(* Logix 5000 project; controller SIMON Emulate 5570 rev 30.12; software revision 30.00 *)

TASK MainTask (periodic, rate 5000 ms, priority 1, watchdog 5000 ms) : MainProgram

MODULES
   Local : Emulate 5570 (ICP 2, rev 30.12)
       : vendor 1 type 0 code 15 (ICP 0, rev 1.1, Output RPI 50 ms)
END_MODULES

TYPE UDT_BA :
STRUCT
   AL : BOOL[128];
END_STRUCT
END_TYPE

PROGRAM MainProgram   (* main routine MainRoutine *)
VAR
   SCAN_CYCLE_TIME : DINT;
   Simon_Ciphertext : DINT[2,2];
   Simon_dec_i : DINT;
   Simon_dec_j : DINT;
   Simon_enc_i : DINT;
   Simon_enc_j : DINT;
   Simon_i : DINT;
   Simon_j : DINT;
   Simon_Plaintext : DINT[2,2];
   Simon_Rd_Max : DINT;
   Simon_Rotate_Result : DINT[2];
   Simon_Round_Keys : DINT[72,2];
   Simon_tmp1 : DINT[2];
   Simon_tmp2 : DINT[2];
   Simon_Ver : DINT;
   Simon_x : DINT[2];
   Simon_y : DINT[2];
END_VAR

ROUTINE MainRoutine   (* ladder *)
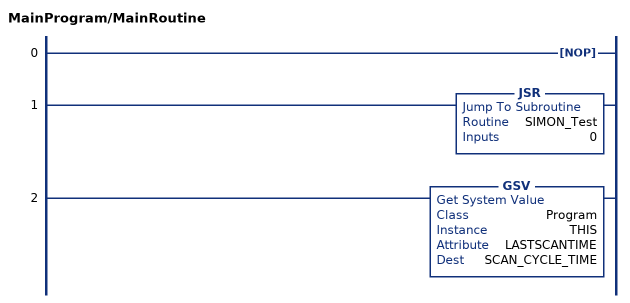
   0: NOP();
   1: JSR(SIMON_Test,0);
   2: GSV(Program,THIS,LASTSCANTIME,SCAN_CYCLE_TIME);
END_ROUTINE

ROUTINE SIMON_ClearKey   (* structured text *)
   Case Simon_Ver Of
   
   0,1,2:
   	For Simon_i:=0 to Simon_Rd_Max by 1 do
   		Simon_Round_Keys[Simon_i,0]:=0;
   	End_For;
   	Simon_tmp1[0]:=0;
   	Simon_tmp2[0]:=0;
   	Simon_Rotate_Result[0]:=0;
   3,4,5:
   	For Simon_i:=0 to Simon_Rd_Max by 1 do
   		Simon_Round_Keys[Simon_i,0]:=0;
   		Simon_Round_Keys[Simon_i,1]:=0;
   	End_For;
   	Simon_tmp1[0]:=0;
   	Simon_tmp1[1]:=0;
   	Simon_tmp2[0]:=0;
   	Simon_tmp2[1]:=0;
   	Simon_Rotate_Result[0]:=0;
   	Simon_Rotate_Result[1]:=0;
   End_Case;
   
   
END_ROUTINE

ROUTINE SIMON_Dec   (* structured text *)
   
   JSR(SIMON_Init);
   
   
   
   
   Case Simon_Ver Of
   
   0,1,2:
   	Simon_Plaintext[1,0]:=Simon_Ciphertext[0,0];
   	Simon_Plaintext[0,0]:=Simon_Ciphertext[1,0];
   
   	For Simon_i:=Simon_Rd_Max to 0 by -1 do
   		Simon_tmp2[0]:=Simon_Plaintext[0,0];  //for rotate
   		JSR(SIMON_Rotate_Left1);	//rotate based on Simon_Ciphertext[0,0]
   		Simon_tmp1[0]:= Simon_Rotate_Result[0];
   		Simon_Rotate_Result[0]:=0;
   
   		Simon_tmp2[0]:=Simon_Plaintext[0,0];  //for rotate
   		JSR(SIMON_Rotate_Left8);
   		Simon_tmp2[0]:=Simon_Rotate_Result[0];
   		Simon_tmp1[0]:= Simon_tmp1[0] AND Simon_tmp2[0];
   		Simon_Rotate_Result[0]:=0;
   
   		Simon_tmp2[0]:=Simon_Plaintext[0,0];  //for rotate
   		JSR(SIMON_Rotate_Left2);
   		Simon_tmp1[0]:= Simon_tmp1[0] XOR Simon_Rotate_Result[0];
   
   		Simon_tmp1[0]:= Simon_tmp1[0] XOR Simon_Round_Keys[Simon_i,0];
   
   		Simon_Plaintext[0,0]:= Simon_Plaintext[1,0] XOR Simon_tmp1[0];
   		Simon_Plaintext[1,0]:= Simon_tmp2[0];
   
   		Simon_Rotate_Result[0]:=0;
   
   	End_for;
   
   3,4,5:
   	Simon_Plaintext[1,0]:=Simon_Ciphertext[0,0];
   	Simon_Plaintext[1,1]:=Simon_Ciphertext[0,1];
   	Simon_Plaintext[0,0]:=Simon_Ciphertext[1,0];
   	Simon_Plaintext[0,1]:=Simon_Ciphertext[1,1];
   
   	For Simon_i:=Simon_Rd_Max to 0 by -1 do
   
   		Simon_tmp2[0]:=Simon_Plaintext[0,0];  //for rotate
   		Simon_tmp2[1]:=Simon_Plaintext[0,1];
   
   		JSR(SIMON_Rotate_Left1);	//rotate based on Simon_Ciphertext[0,0] and [0,1]
   		Simon_tmp1[0]:= Simon_Rotate_Result[0];
   		Simon_tmp1[1]:= Simon_Rotate_Result[1];
   
   		Simon_Rotate_Result[0]:=0;
   		Simon_Rotate_Result[1]:=0;
   
   		Simon_tmp2[0]:=Simon_Plaintext[0,0];
   		Simon_tmp2[1]:=Simon_Plaintext[0,1];
   		JSR(SIMON_Rotate_Left8);
   		Simon_tmp2[0]:=Simon_Rotate_Result[0];
   		Simon_tmp2[1]:=Simon_Rotate_Result[1];
   		Simon_tmp1[0]:= Simon_tmp1[0] AND Simon_tmp2[0];
   		Simon_tmp1[1]:= Simon_tmp1[1] AND Simon_tmp2[1];
   
   		Simon_tmp2[0]:=Simon_Plaintext[0,0];
   		Simon_tmp2[1]:=Simon_Plaintext[0,1];
   
   		Simon_Rotate_Result[0]:=0;
   		Simon_Rotate_Result[1]:=0;
   
   		JSR(SIMON_Rotate_Left2);
   		Simon_tmp1[0]:= Simon_tmp1[0] XOR Simon_Rotate_Result[0];
   		Simon_tmp1[1]:= Simon_tmp1[1] XOR Simon_Rotate_Result[1];
   
   		Simon_tmp1[0]:= Simon_tmp1[0] XOR Simon_Round_Keys[Simon_i,0];
   		Simon_tmp1[1]:= Simon_tmp1[1] XOR Simon_Round_Keys[Simon_i,1];
   
   
   		Simon_Plaintext[0,0]:= Simon_Plaintext[1,0] XOR Simon_tmp1[0];
   		Simon_Plaintext[0,1]:= Simon_Plaintext[1,1] XOR Simon_tmp1[1];
   
   		Simon_Plaintext[1,0]:= Simon_tmp2[0];
   		Simon_Plaintext[1,1]:= Simon_tmp2[1];
   
   		Simon_Rotate_Result[0]:=0;
   		Simon_Rotate_Result[1]:=0;
   
   	End_for;
   
   End_Case;
   
   
   
   
   
   
   JSR(SIMON_ClearKey);
   
   
   
   
   
   
   
   
END_ROUTINE

ROUTINE SIMON_Enc   (* structured text *)
   
   JSR(SIMON_Init);
   
   
   
   
   
   Case Simon_Ver Of
   
   0,1,2:
   	//Simon_Ciphertext[1,0]:=Simon_Plaintext[0,0];
   	//Simon_Ciphertext[0,0]:=Simon_Plaintext[1,0];
   
   	Simon_Ciphertext[0,0]:=Simon_Plaintext[1,0];
   	Simon_Ciphertext[1,0]:=Simon_Plaintext[0,0];
   
   	For Simon_i:=0 to Simon_Rd_Max by 1 do
   		Simon_tmp2[0]:=Simon_Ciphertext[0,0];  //for rotate
   		JSR(SIMON_Rotate_Left1);	//rotate based on Simon_Plaintext[0,0]
   		Simon_tmp1[0]:= Simon_Rotate_Result[0];
   		Simon_Rotate_Result[0]:=0;
   
   		Simon_tmp2[0]:=Simon_Ciphertext[0,0];  //for rotate
   		JSR(SIMON_Rotate_Left8);
   		Simon_tmp2[0]:=Simon_Rotate_Result[0];
   
   		Simon_tmp1[0]:= Simon_tmp1[0] AND Simon_tmp2[0];
   		Simon_Rotate_Result[0]:=0;
   
   		Simon_tmp2[0]:=Simon_Ciphertext[0,0];  //for rotate
   		JSR(SIMON_Rotate_Left2);
   		Simon_tmp1[0]:= Simon_tmp1[0] XOR Simon_Rotate_Result[0];
   
   		Simon_tmp1[0]:= Simon_tmp1[0] XOR Simon_Round_Keys[Simon_i,0];
   
   		Simon_Ciphertext[0,0]:= Simon_Ciphertext[1,0] XOR Simon_tmp1[0];
   		Simon_Ciphertext[1,0]:= Simon_tmp2[0];
   
   		Simon_Rotate_Result[0]:=0;
   
   	End_for;
   
   3,4,5:
   	Simon_Ciphertext[1,0]:=Simon_Plaintext[0,0];
   	Simon_Ciphertext[1,1]:=Simon_Plaintext[0,1];
   	Simon_Ciphertext[0,0]:=Simon_Plaintext[1,0];
   	Simon_Ciphertext[0,1]:=Simon_Plaintext[1,1];
   
   	For Simon_i:=0 to Simon_Rd_Max by 1 do
   
   		Simon_tmp2[0]:=Simon_Ciphertext[0,0];  //for rotate
   		Simon_tmp2[1]:=Simon_Ciphertext[0,1];
   
   		JSR(SIMON_Rotate_Left1);	//rotate based on Simon_Plaintext[0,0] and [0,1]
   		Simon_tmp1[0]:= Simon_Rotate_Result[0];
   		Simon_tmp1[1]:= Simon_Rotate_Result[1];
   
   		Simon_Rotate_Result[0]:=0;
   		Simon_Rotate_Result[1]:=0;
   
   		Simon_tmp2[0]:=Simon_Ciphertext[0,0];
   		Simon_tmp2[1]:=Simon_Ciphertext[0,1];
   		JSR(SIMON_Rotate_Left8);
   		Simon_tmp2[0]:=Simon_Rotate_Result[0];
   		Simon_tmp2[1]:=Simon_Rotate_Result[1];
   		Simon_tmp1[0]:= Simon_tmp1[0] AND Simon_tmp2[0];
   		Simon_tmp1[1]:= Simon_tmp1[1] AND Simon_tmp2[1];
   
   		Simon_Rotate_Result[0]:=0;
   		Simon_Rotate_Result[1]:=0;
   
   		Simon_tmp2[0]:=Simon_Ciphertext[0,0];
   		Simon_tmp2[1]:=Simon_Ciphertext[0,1];
   		JSR(SIMON_Rotate_Left2);
   		Simon_tmp1[0]:= Simon_tmp1[0] XOR Simon_Rotate_Result[0];
   		Simon_tmp1[1]:= Simon_tmp1[1] XOR Simon_Rotate_Result[1];
   
   		Simon_tmp1[0]:= Simon_tmp1[0] XOR Simon_Round_Keys[Simon_i,0];
   		Simon_tmp1[1]:= Simon_tmp1[1] XOR Simon_Round_Keys[Simon_i,1];
   
   
   		Simon_Ciphertext[0,0]:= Simon_Ciphertext[1,0] XOR Simon_tmp1[0];
   		Simon_Ciphertext[0,1]:= Simon_Ciphertext[1,1] XOR Simon_tmp1[1];
   
   		Simon_Ciphertext[1,0]:= Simon_tmp2[0];
   		Simon_Ciphertext[1,1]:= Simon_tmp2[1];
   
   		Simon_Rotate_Result[0]:=0;
   		Simon_Rotate_Result[1]:=0;
   
   	End_for;
   
   End_Case;
   
   
   
   
   
   JSR(SIMON_ClearKey);
   
   
   
   
   
   
END_ROUTINE

ROUTINE SIMON_Init   (* structured text *)
   CASE Simon_Ver Of
   	0:
   		Simon_Rd_Max:=31;
   		Simon_Round_Keys[0,0]:=256;
   		Simon_Round_Keys[1,0]:=2312;
   		Simon_Round_Keys[2,0]:=4368;
   		Simon_Round_Keys[3,0]:=6424;
   		Simon_Round_Keys[4,0]:=29123;
   		Simon_Round_Keys[5,0]:=46665;
   		Simon_Round_Keys[6,0]:=22228;
   		Simon_Round_Keys[7,0]:=57456;
   		Simon_Round_Keys[8,0]:=61786;
   		Simon_Round_Keys[9,0]:=50485;
   		Simon_Round_Keys[10,0]:=56724;
   		Simon_Round_Keys[11,0]:=16400;
   		Simon_Round_Keys[12,0]:=9482;
   		Simon_Round_Keys[13,0]:=28518;
   		Simon_Round_Keys[14,0]:=59755;
   		Simon_Round_Keys[15,0]:=19416;
   		Simon_Round_Keys[16,0]:=4069;
   		Simon_Round_Keys[17,0]:=31815;
   		Simon_Round_Keys[18,0]:=57583;
   		Simon_Round_Keys[19,0]:=15905;
   		Simon_Round_Keys[20,0]:=1627;
   		Simon_Round_Keys[21,0]:=17292;
   		Simon_Round_Keys[22,0]:=62058;
   		Simon_Round_Keys[23,0]:=46528;
   		Simon_Round_Keys[24,0]:=34313;
   		Simon_Round_Keys[25,0]:=40846;
   		Simon_Round_Keys[26,0]:=55487;
   		Simon_Round_Keys[27,0]:=2476;
   		Simon_Round_Keys[28,0]:=59410;
   		Simon_Round_Keys[29,0]:=10000;
   		Simon_Round_Keys[30,0]:=11434;
   		Simon_Round_Keys[31,0]:=36116;
   
   	1:
   		Simon_Rd_Max:=41;
   		Simon_Round_Keys[0,0]:=50462976;
   		Simon_Round_Keys[1,0]:=185207048;
   		Simon_Round_Keys[2,0]:=319951120;
   		Simon_Round_Keys[3,0]:=-5333554;
   		Simon_Round_Keys[4,0]:=-990196591;
   		Simon_Round_Keys[5,0]:=-935519306;
   		Simon_Round_Keys[6,0]:=-1244327681;
   		Simon_Round_Keys[7,0]:=920830076;
   		Simon_Round_Keys[8,0]:=1919979587;
   		Simon_Round_Keys[9,0]:=323220494;
   		Simon_Round_Keys[10,0]:=-364806592;
   		Simon_Round_Keys[11,0]:=-1637656685;
   		Simon_Round_Keys[12,0]:=-1500097416;
   		Simon_Round_Keys[13,0]:=-1962594699;
   		Simon_Round_Keys[14,0]:=-2008260793;
   		Simon_Round_Keys[15,0]:=-790305384;
   		Simon_Round_Keys[16,0]:=-471334045;
   		Simon_Round_Keys[17,0]:=904929505;
   		Simon_Round_Keys[18,0]:=452598902;
   		Simon_Round_Keys[19,0]:=-1092149546;
   		Simon_Round_Keys[20,0]:=1983728938;
   		Simon_Round_Keys[21,0]:=211918588;
   		Simon_Round_Keys[22,0]:=4639515;
   		Simon_Round_Keys[23,0]:=1506674436;
   		Simon_Round_Keys[24,0]:=1039876497;
   		Simon_Round_Keys[25,0]:=-874911540;
   		Simon_Round_Keys[26,0]:=-201893011;
   		Simon_Round_Keys[27,0]:=-1555750729;
   		Simon_Round_Keys[28,0]:=-1166352083;
   		Simon_Round_Keys[29,0]:=1625314982;
   		Simon_Round_Keys[30,0]:=-156708620;
   		Simon_Round_Keys[31,0]:=-1808102975;
   		Simon_Round_Keys[32,0]:=-1260695298;
   		Simon_Round_Keys[33,0]:=880930840;
   		Simon_Round_Keys[34,0]:=-300067009;
   		Simon_Round_Keys[35,0]:=1208406167;
   		Simon_Round_Keys[36,0]:=1459534079;
   		Simon_Round_Keys[37,0]:=240292946;
   		Simon_Round_Keys[38,0]:=-690596700;
   		Simon_Round_Keys[39,0]:=2125916381;
   		Simon_Round_Keys[40,0]:=-1986996168;
   		Simon_Round_Keys[41,0]:=-1333608996;
   	2:
   		Simon_Rd_Max:=43;
   		Simon_Round_Keys[0,0]:=50462976;
   		Simon_Round_Keys[1,0]:=185207048;
   		Simon_Round_Keys[2,0]:=319951120;
   		Simon_Round_Keys[3,0]:=454695192;
   		Simon_Round_Keys[4,0]:=1889538499;
   		Simon_Round_Keys[5,0]:=-1217336247;
   		Simon_Round_Keys[6,0]:=1474553909;
   		Simon_Round_Keys[7,0]:=-745030590;
   		Simon_Round_Keys[8,0]:=-1797457889;
   		Simon_Round_Keys[9,0]:=-1085579496;
   		Simon_Round_Keys[10,0]:=-1906463815;
   		Simon_Round_Keys[11,0]:=-604723101;
   		Simon_Round_Keys[12,0]:=-854841092;
   		Simon_Round_Keys[13,0]:=1555470609;
   		Simon_Round_Keys[14,0]:=2045842085;
   		Simon_Round_Keys[15,0]:=1998608483;
   		Simon_Round_Keys[16,0]:=-1719137262;
   		Simon_Round_Keys[17,0]:=485063768;
   		Simon_Round_Keys[18,0]:=-923983547;
   		Simon_Round_Keys[19,0]:=-1207903304;
   		Simon_Round_Keys[20,0]:=-395696298;
   		Simon_Round_Keys[21,0]:=2080822493;
   		Simon_Round_Keys[22,0]:=-1420632310;
   		Simon_Round_Keys[23,0]:=612329128;
   		Simon_Round_Keys[24,0]:=1398308006;
   		Simon_Round_Keys[25,0]:=-765717519;
   		Simon_Round_Keys[26,0]:=1166259787;
   		Simon_Round_Keys[27,0]:=2107414029;
   		Simon_Round_Keys[28,0]:=-272645389;
   		Simon_Round_Keys[29,0]:=-1980922605;
   		Simon_Round_Keys[30,0]:=814611534;
   		Simon_Round_Keys[31,0]:=-1088804298;
   		Simon_Round_Keys[32,0]:=-515269264;
   		Simon_Round_Keys[33,0]:=1290064639;
   		Simon_Round_Keys[34,0]:=850914287;
   		Simon_Round_Keys[35,0]:=-998963775;
   		Simon_Round_Keys[36,0]:=-790025752;
   		Simon_Round_Keys[37,0]:=-1880849223;
   		Simon_Round_Keys[38,0]:=1107643374;
   		Simon_Round_Keys[39,0]:=-1351107870;
   		Simon_Round_Keys[40,0]:=404331522;
   		Simon_Round_Keys[41,0]:=1906196252;
   		Simon_Round_Keys[42,0]:=203224979;
   		Simon_Round_Keys[43,0]:=366954134;
   	3:
   		Simon_Rd_Max:=67;
   		Simon_Round_Keys[0,0]:=50462976;
   		Simon_Round_Keys[0,1]:=117835012;
   		Simon_Round_Keys[1,0]:=185207048;
   		Simon_Round_Keys[1,1]:=252579084;
   		Simon_Round_Keys[2,0]:=-1121181876;
   		Simon_Round_Keys[2,1]:=2045303690;
   		Simon_Round_Keys[3,0]:=142783721;
   		Simon_Round_Keys[3,1]:=-1202559942;
   		Simon_Round_Keys[4,0]:=-1555325598;
   		Simon_Round_Keys[4,1]:=714624689;
   		Simon_Round_Keys[5,0]:=-652181137;
   		Simon_Round_Keys[5,1]:=542578424;
   		Simon_Round_Keys[6,0]:=-905807196;
   		Simon_Round_Keys[6,1]:=-1016585474;
   		Simon_Round_Keys[7,0]:=322901612;
   		Simon_Round_Keys[7,1]:=200503159;
   		Simon_Round_Keys[8,0]:=-1498835214;
   		Simon_Round_Keys[8,1]:=2102822424;
   		Simon_Round_Keys[9,0]:=1920942624;
   		Simon_Round_Keys[9,1]:=-1670174678;
   		Simon_Round_Keys[10,0]:=-1338083992;
   		Simon_Round_Keys[10,1]:=-1730138528;
   		Simon_Round_Keys[11,0]:=-1870359514;
   		Simon_Round_Keys[11,1]:=-115420929;
   		Simon_Round_Keys[12,0]:=1155092819;
   		Simon_Round_Keys[12,1]:=-676469105;
   		Simon_Round_Keys[13,0]:=1940772068;
   		Simon_Round_Keys[13,1]:=1097747897;
   		Simon_Round_Keys[14,0]:=40487293;
   		Simon_Round_Keys[14,1]:=-462867428;
   		Simon_Round_Keys[15,0]:=-868643168;
   		Simon_Round_Keys[15,1]:=-598079612;
   		Simon_Round_Keys[16,0]:=684892095;
   		Simon_Round_Keys[16,1]:=232270699;
   		Simon_Round_Keys[17,0]:=-464450736;
   		Simon_Round_Keys[17,1]:=851672992;
   		Simon_Round_Keys[18,0]:=-975023716;
   		Simon_Round_Keys[18,1]:=-145519462;
   		Simon_Round_Keys[19,0]:=-280192122;
   		Simon_Round_Keys[19,1]:=-1666987771;
   		Simon_Round_Keys[20,0]:=-654248791;
   		Simon_Round_Keys[20,1]:=-1292749099;
   		Simon_Round_Keys[21,0]:=-167545436;
   		Simon_Round_Keys[21,1]:=-835890355;
   		Simon_Round_Keys[22,0]:=1197429435;
   		Simon_Round_Keys[22,1]:=-1742031241;
   		Simon_Round_Keys[23,0]:=-1788701403;
   		Simon_Round_Keys[23,1]:=-78294757;
   		Simon_Round_Keys[24,0]:=1935333041;
   		Simon_Round_Keys[24,1]:=-2029340998;
   		Simon_Round_Keys[25,0]:=-2084332188;
   		Simon_Round_Keys[25,1]:=742085464;
   		Simon_Round_Keys[26,0]:=350315318;
   		Simon_Round_Keys[26,1]:=-1078880741;
   		Simon_Round_Keys[27,0]:=-1343334195;
   		Simon_Round_Keys[27,1]:=1875478277;
   		Simon_Round_Keys[28,0]:=69055071;
   		Simon_Round_Keys[28,1]:=994820468;
   		Simon_Round_Keys[29,0]:=-1865168290;
   		Simon_Round_Keys[29,1]:=-2064925501;
   		Simon_Round_Keys[30,0]:=-1326118836;
   		Simon_Round_Keys[30,1]:=-60296481;
   		Simon_Round_Keys[31,0]:=1648215087;
   		Simon_Round_Keys[31,1]:=727630410;
   		Simon_Round_Keys[32,0]:=-1519479945;
   		Simon_Round_Keys[32,1]:=340146509;
   		Simon_Round_Keys[33,0]:=-214368118;
   		Simon_Round_Keys[33,1]:=1198364936;
   		Simon_Round_Keys[34,0]:=-876225389;
   		Simon_Round_Keys[34,1]:=119712771;
   		Simon_Round_Keys[35,0]:=1224874285;
   		Simon_Round_Keys[35,1]:=-402384457;
   		Simon_Round_Keys[36,0]:=-1450556967;
   		Simon_Round_Keys[36,1]:=-1688366767;
   		Simon_Round_Keys[37,0]:=-1722545417;
   		Simon_Round_Keys[37,1]:=-1121612425;
   		Simon_Round_Keys[38,0]:=-590708780;
   		Simon_Round_Keys[38,1]:=-388724777;
   		Simon_Round_Keys[39,0]:=-520217332;
   		Simon_Round_Keys[39,1]:=-1857181169;
   		Simon_Round_Keys[40,0]:=556114521;
   		Simon_Round_Keys[40,1]:=1276516297;
   		Simon_Round_Keys[41,0]:=-1456010081;
   		Simon_Round_Keys[41,1]:=-739117451;
   		Simon_Round_Keys[42,0]:=829410559;
   		Simon_Round_Keys[42,1]:=-1264006753;
   		Simon_Round_Keys[43,0]:=1140061747;
   		Simon_Round_Keys[43,1]:=567385120;
   		Simon_Round_Keys[44,0]:=-1026461018;
   		Simon_Round_Keys[44,1]:=493886502;
   		Simon_Round_Keys[45,0]:=142291120;
   		Simon_Round_Keys[45,1]:=2086101401;
   		Simon_Round_Keys[46,0]:=-1935255482;
   		Simon_Round_Keys[46,1]:=-356484621;
   		Simon_Round_Keys[47,0]:=-1092984383;
   		Simon_Round_Keys[47,1]:=811374279;
   		Simon_Round_Keys[48,0]:=-9482849;
   		Simon_Round_Keys[48,1]:=540138936;
   		Simon_Round_Keys[49,0]:=-784432298;
   		Simon_Round_Keys[49,1]:=-643412140;
   		Simon_Round_Keys[50,0]:=-677082563;
   		Simon_Round_Keys[50,1]:=1767935832;
   		Simon_Round_Keys[51,0]:=-1185962674;
   		Simon_Round_Keys[51,1]:=1575201205;
   		Simon_Round_Keys[52,0]:=-991528132;
   		Simon_Round_Keys[52,1]:=-1191362806;
   		Simon_Round_Keys[53,0]:=-1302138265;
   		Simon_Round_Keys[53,1]:=-24370597;
   		Simon_Round_Keys[54,0]:=-160172630;
   		Simon_Round_Keys[54,1]:=-952400229;
   		Simon_Round_Keys[55,0]:=-1942729611;
   		Simon_Round_Keys[55,1]:=-169405154;
   		Simon_Round_Keys[56,0]:=818530078;
   		Simon_Round_Keys[56,1]:=-651761002;
   		Simon_Round_Keys[57,0]:=-690088165;
   		Simon_Round_Keys[57,1]:=1018059034;
   		Simon_Round_Keys[58,0]:=947919729;
   		Simon_Round_Keys[58,1]:=-226083877;
   		Simon_Round_Keys[59,0]:=-38147521;
   		Simon_Round_Keys[59,1]:=-500628957;
   		Simon_Round_Keys[60,0]:=-2028779671;
   		Simon_Round_Keys[60,1]:=253654082;
   		Simon_Round_Keys[61,0]:=2060798296;
   		Simon_Round_Keys[61,1]:=-1396386800;
   		Simon_Round_Keys[62,0]:=1880835370;
   		Simon_Round_Keys[62,1]:=1874156670;
   		Simon_Round_Keys[63,0]:=-1406637486;
   		Simon_Round_Keys[63,1]:=-1204365913;
   		Simon_Round_Keys[64,0]:=10694968;
   		Simon_Round_Keys[64,1]:=-321973137;
   		Simon_Round_Keys[65,0]:=1137295514;
   		Simon_Round_Keys[65,1]:=-727959149;
   		Simon_Round_Keys[66,0]:=-1558615329;
   		Simon_Round_Keys[66,1]:=-454381765;
   		Simon_Round_Keys[67,0]:=1919190160;
   		Simon_Round_Keys[67,1]:=699414904;
   	4:
   		Simon_Rd_Max:=68;
   		Simon_Round_Keys[0,0]:=50462976;
   		Simon_Round_Keys[0,1]:=117835012;
   		Simon_Round_Keys[1,0]:=185207048;
   		Simon_Round_Keys[1,1]:=252579084;
   		Simon_Round_Keys[2,0]:=319951120;
   		Simon_Round_Keys[2,1]:=387323156;
   		Simon_Round_Keys[3,0]:=1068408270;
   		Simon_Round_Keys[3,1]:=-76916472;
   		Simon_Round_Keys[4,0]:=1895484560;
   		Simon_Round_Keys[4,1]:=-1070982078;
   		Simon_Round_Keys[5,0]:=-2047009865;
   		Simon_Round_Keys[5,1]:=-51509081;
   		Simon_Round_Keys[6,0]:=1219563774;
   		Simon_Round_Keys[6,1]:=-2067363991;
   		Simon_Round_Keys[7,0]:=848822397;
   		Simon_Round_Keys[7,1]:=117529382;
   		Simon_Round_Keys[8,0]:=-545758141;
   		Simon_Round_Keys[8,1]:=1937885582;
   		Simon_Round_Keys[9,0]:=-2125044273;
   		Simon_Round_Keys[9,1]:=577854783;
   		Simon_Round_Keys[10,0]:=-984066715;
   		Simon_Round_Keys[10,1]:=-292054355;
   		Simon_Round_Keys[11,0]:=1148785732;
   		Simon_Round_Keys[11,1]:=1866841230;
   		Simon_Round_Keys[12,0]:=1382099455;
   		Simon_Round_Keys[12,1]:=378687129;
   		Simon_Round_Keys[13,0]:=-2050122440;
   		Simon_Round_Keys[13,1]:=47384680;
   		Simon_Round_Keys[14,0]:=593723852;
   		Simon_Round_Keys[14,1]:=281875194;
   		Simon_Round_Keys[15,0]:=1271176743;
   		Simon_Round_Keys[15,1]:=-1434926570;
   		Simon_Round_Keys[16,0]:=-671696669;
   		Simon_Round_Keys[16,1]:=1925473268;
   		Simon_Round_Keys[17,0]:=186499746;
   		Simon_Round_Keys[17,1]:=-1236916412;
   		Simon_Round_Keys[18,0]:=1978205605;
   		Simon_Round_Keys[18,1]:=673946485;
   		Simon_Round_Keys[19,0]:=-773130255;
   		Simon_Round_Keys[19,1]:=2059163346;
   		Simon_Round_Keys[20,0]:=-2084451106;
   		Simon_Round_Keys[20,1]:=1900386060;
   		Simon_Round_Keys[21,0]:=-766320882;
   		Simon_Round_Keys[21,1]:=-18313445;
   		Simon_Round_Keys[22,0]:=-377848292;
   		Simon_Round_Keys[22,1]:=-1250938817;
   		Simon_Round_Keys[23,0]:=2139544320;
   		Simon_Round_Keys[23,1]:=-750555657;
   		Simon_Round_Keys[24,0]:=-1247439325;
   		Simon_Round_Keys[24,1]:=374025093;
   		Simon_Round_Keys[25,0]:=-76846522;
   		Simon_Round_Keys[25,1]:=421664776;
   		Simon_Round_Keys[26,0]:=279117585;
   		Simon_Round_Keys[26,1]:=-1911885687;
   		Simon_Round_Keys[27,0]:=-112977459;
   		Simon_Round_Keys[27,1]:=-1063967389;
   		Simon_Round_Keys[28,0]:=1143494430;
   		Simon_Round_Keys[28,1]:=-2100948723;
   		Simon_Round_Keys[29,0]:=-1818587266;
   		Simon_Round_Keys[29,1]:=1233235015;
   		Simon_Round_Keys[30,0]:=-1913577687;
   		Simon_Round_Keys[30,1]:=314766800;
   		Simon_Round_Keys[31,0]:=-1565091083;
   		Simon_Round_Keys[31,1]:=-833773803;
   		Simon_Round_Keys[32,0]:=-2112304525;
   		Simon_Round_Keys[32,1]:=1397963179;
   		Simon_Round_Keys[33,0]:=-1167297220;
   		Simon_Round_Keys[33,1]:=-1302176128;
   		Simon_Round_Keys[34,0]:=1101147389;
   		Simon_Round_Keys[34,1]:=1826098898;
   		Simon_Round_Keys[35,0]:=298406623;
   		Simon_Round_Keys[35,1]:=-671463581;
   		Simon_Round_Keys[36,0]:=381040055;
   		Simon_Round_Keys[36,1]:=1243434469;
   		Simon_Round_Keys[37,0]:=1306556140;
   		Simon_Round_Keys[37,1]:=247827535;
   		Simon_Round_Keys[38,0]:=-212556656;
   		Simon_Round_Keys[38,1]:=1764839889;
   		Simon_Round_Keys[39,0]:=-938077039;
   		Simon_Round_Keys[39,1]:=-1101558467;
   		Simon_Round_Keys[40,0]:=-677631285;
   		Simon_Round_Keys[40,1]:=-585762108;
   		Simon_Round_Keys[41,0]:=-618586983;
   		Simon_Round_Keys[41,1]:=1354583770;
   		Simon_Round_Keys[42,0]:=-1052780233;
   		Simon_Round_Keys[42,1]:=-21753868;
   		Simon_Round_Keys[43,0]:=-61353085;
   		Simon_Round_Keys[43,1]:=-1562917830;
   		Simon_Round_Keys[44,0]:=-728669139;
   		Simon_Round_Keys[44,1]:=-516606495;
   		Simon_Round_Keys[45,0]:=421207053;
   		Simon_Round_Keys[45,1]:=1669203433;
   		Simon_Round_Keys[46,0]:=-1323631042;
   		Simon_Round_Keys[46,1]:=661658406;
   		Simon_Round_Keys[47,0]:=-1772327947;
   		Simon_Round_Keys[47,1]:=945014984;
   		Simon_Round_Keys[48,0]:=2102044721;
   		Simon_Round_Keys[48,1]:=1745796995;
   		Simon_Round_Keys[49,0]:=379125318;
   		Simon_Round_Keys[49,1]:=-485566255;
   		Simon_Round_Keys[50,0]:=1511588900;
   		Simon_Round_Keys[50,1]:=1979515296;
   		Simon_Round_Keys[51,0]:=-1940396277;
   		Simon_Round_Keys[51,1]:=1578184786;
   		Simon_Round_Keys[52,0]:=-1876393173;
   		Simon_Round_Keys[52,1]:=-1026420191;
   		Simon_Round_Keys[53,0]:=-1897831538;
   		Simon_Round_Keys[53,1]:=1316330809;
   		Simon_Round_Keys[54,0]:=-627432769;
   		Simon_Round_Keys[54,1]:=-1933105703;
   		Simon_Round_Keys[55,0]:=-919758165;
   		Simon_Round_Keys[55,1]:=880376632;
   		Simon_Round_Keys[56,0]:=-458623348;
   		Simon_Round_Keys[56,1]:=1682102802;
   		Simon_Round_Keys[57,0]:=1471839482;
   		Simon_Round_Keys[57,1]:=972336325;
   		Simon_Round_Keys[58,0]:=-916550393;
   		Simon_Round_Keys[58,1]:=791108499;
   		Simon_Round_Keys[59,0]:=1592274944;
   		Simon_Round_Keys[59,1]:=212581158;
   		Simon_Round_Keys[60,0]:=108398086;
   		Simon_Round_Keys[60,1]:=-950755348;
   		Simon_Round_Keys[61,0]:=1980289626;
   		Simon_Round_Keys[61,1]:=1682407023;
   		Simon_Round_Keys[62,0]:=-1196009325;
   		Simon_Round_Keys[62,1]:=429448434;
   		Simon_Round_Keys[63,0]:=-2062264480;
   		Simon_Round_Keys[63,1]:=1778513474;
   		Simon_Round_Keys[64,0]:=-251338179;
   		Simon_Round_Keys[64,1]:=-1873240004;
   		Simon_Round_Keys[65,0]:=377058570;
   		Simon_Round_Keys[65,1]:=-1922450167;
   		Simon_Round_Keys[66,0]:=-918351508;
   		Simon_Round_Keys[66,1]:=1820698060;
   		Simon_Round_Keys[67,0]:=1531399930;
   		Simon_Round_Keys[67,1]:=620736806;
   		Simon_Round_Keys[68,0]:=1197086663;
   		Simon_Round_Keys[68,1]:=-1807331392;
   	5:
   		Simon_Rd_Max:=71;
   		Simon_Round_Keys[0,0]:=50462976;
   		Simon_Round_Keys[0,1]:=117835012;
   		Simon_Round_Keys[1,0]:=185207048;
   		Simon_Round_Keys[1,1]:=252579084;
   		Simon_Round_Keys[2,0]:=319951120;
   		Simon_Round_Keys[2,1]:=387323156;
   		Simon_Round_Keys[3,0]:=454695192;
   		Simon_Round_Keys[3,1]:=522067228;
   		Simon_Round_Keys[4,0]:=-1331686973;
   		Simon_Round_Keys[4,1]:=1919079171;
   		Simon_Round_Keys[5,0]:=-1552880567;
   		Simon_Round_Keys[5,1]:=-1257858499;
   		Simon_Round_Keys[6,0]:=-1809586123;
   		Simon_Round_Keys[6,1]:=1434993565;
   		Simon_Round_Keys[7,0]:=-405554110;
   		Simon_Round_Keys[7,1]:=-732179413;
   		Simon_Round_Keys[8,0]:=-15714274;
   		Simon_Round_Keys[8,1]:=-1781122024;
   		Simon_Round_Keys[9,0]:=-1834087656;
   		Simon_Round_Keys[9,1]:=-1907186733;
   		Simon_Round_Keys[10,0]:=882463864;
   		Simon_Round_Keys[10,1]:=-1926300645;
   		Simon_Round_Keys[11,0]:=1299109990;
   		Simon_Round_Keys[11,1]:=1844328834;
   		Simon_Round_Keys[12,0]:=913178621;
   		Simon_Round_Keys[12,1]:=137434485;
   		Simon_Round_Keys[13,0]:=909077153;
   		Simon_Round_Keys[13,1]:=-879628861;
   		Simon_Round_Keys[14,0]:=-182975442;
   		Simon_Round_Keys[14,1]:=201524675;
   		Simon_Round_Keys[15,0]:=1580771166;
   		Simon_Round_Keys[15,1]:=1064831318;
   		Simon_Round_Keys[16,0]:=-896646802;
   		Simon_Round_Keys[16,1]:=-40931305;
   		Simon_Round_Keys[17,0]:=1136508766;
   		Simon_Round_Keys[17,1]:=235244573;
   		Simon_Round_Keys[18,0]:=126837564;
   		Simon_Round_Keys[18,1]:=-233300349;
   		Simon_Round_Keys[19,0]:=-561568977;
   		Simon_Round_Keys[19,1]:=313375885;
   		Simon_Round_Keys[20,0]:=-1322629067;
   		Simon_Round_Keys[20,1]:=403220898;
   		Simon_Round_Keys[21,0]:=1161658245;
   		Simon_Round_Keys[21,1]:=-2005926514;
   		Simon_Round_Keys[22,0]:=-448768399;
   		Simon_Round_Keys[22,1]:=2140636126;
   		Simon_Round_Keys[23,0]:=-96747692;
   		Simon_Round_Keys[23,1]:=1096103495;
   		Simon_Round_Keys[24,0]:=-1450001519;
   		Simon_Round_Keys[24,1]:=1737531576;
   		Simon_Round_Keys[25,0]:=-1299611142;
   		Simon_Round_Keys[25,1]:=-1924702628;
   		Simon_Round_Keys[26,0]:=1088446802;
   		Simon_Round_Keys[26,1]:=418074475;
   		Simon_Round_Keys[27,0]:=613264590;
   		Simon_Round_Keys[27,1]:=140633159;
   		Simon_Round_Keys[28,0]:=729377343;
   		Simon_Round_Keys[28,1]:=1912704249;
   		Simon_Round_Keys[29,0]:=440308761;
   		Simon_Round_Keys[29,1]:=2135318573;
   		Simon_Round_Keys[30,0]:=2066800580;
   		Simon_Round_Keys[30,1]:=1398344951;
   		Simon_Round_Keys[31,0]:=-43869674;
   		Simon_Round_Keys[31,1]:=-205397908;
   		Simon_Round_Keys[32,0]:=333263157;
   		Simon_Round_Keys[32,1]:=-60882634;
   		Simon_Round_Keys[33,0]:=-2144358666;
   		Simon_Round_Keys[33,1]:=436340075;
   		Simon_Round_Keys[34,0]:=-820250604;
   		Simon_Round_Keys[34,1]:=-2073590871;
   		Simon_Round_Keys[35,0]:=-1111749434;
   		Simon_Round_Keys[35,1]:=-695986575;
   		Simon_Round_Keys[36,0]:=-2139687408;
   		Simon_Round_Keys[36,1]:=-1558496578;
   		Simon_Round_Keys[37,0]:=1867506870;
   		Simon_Round_Keys[37,1]:=1039887381;
   		Simon_Round_Keys[38,0]:=-1466232944;
   		Simon_Round_Keys[38,1]:=1648278108;
   		Simon_Round_Keys[39,0]:=-577458392;
   		Simon_Round_Keys[39,1]:=-779521407;
   		Simon_Round_Keys[40,0]:=-2130001897;
   		Simon_Round_Keys[40,1]:=-389306842;
   		Simon_Round_Keys[41,0]:=-732469488;
   		Simon_Round_Keys[41,1]:=313571902;
   		Simon_Round_Keys[42,0]:=1408602691;
   		Simon_Round_Keys[42,1]:=670143110;
   		Simon_Round_Keys[43,0]:=1285888932;
   		Simon_Round_Keys[43,1]:=1683608371;
   		Simon_Round_Keys[44,0]:=-1646847555;
   		Simon_Round_Keys[44,1]:=-971892307;
   		Simon_Round_Keys[45,0]:=1002459426;
   		Simon_Round_Keys[45,1]:=1038449835;
   		Simon_Round_Keys[46,0]:=-1841695490;
   		Simon_Round_Keys[46,1]:=-367415412;
   		Simon_Round_Keys[47,0]:=-1157443350;
   		Simon_Round_Keys[47,1]:=-1923115330;
   		Simon_Round_Keys[48,0]:=-120002335;
   		Simon_Round_Keys[48,1]:=-477876464;
   		Simon_Round_Keys[49,0]:=260846541;
   		Simon_Round_Keys[49,1]:=2135374861;
   		Simon_Round_Keys[50,0]:=-95619367;
   		Simon_Round_Keys[50,1]:=-1509254701;
   		Simon_Round_Keys[51,0]:=-2136677839;
   		Simon_Round_Keys[51,1]:=-834163842;
   		Simon_Round_Keys[52,0]:=-1217138862;
   		Simon_Round_Keys[52,1]:=-105644740;
   		Simon_Round_Keys[53,0]:=-1434451301;
   		Simon_Round_Keys[53,1]:=-2061871428;
   		Simon_Round_Keys[54,0]:=-1698850186;
   		Simon_Round_Keys[54,1]:=-1201408175;
   		Simon_Round_Keys[55,0]:=-1184010274;
   		Simon_Round_Keys[55,1]:=139990716;
   		Simon_Round_Keys[56,0]:=-336107394;
   		Simon_Round_Keys[56,1]:=1616247965;
   		Simon_Round_Keys[57,0]:=1633497506;
   		Simon_Round_Keys[57,1]:=-1262991904;
   		Simon_Round_Keys[58,0]:=-1968715628;
   		Simon_Round_Keys[58,1]:=909416878;
   		Simon_Round_Keys[59,0]:=1633733113;
   		Simon_Round_Keys[59,1]:=1652371775;
   		Simon_Round_Keys[60,0]:=1606495056;
   		Simon_Round_Keys[60,1]:=-886697658;
   		Simon_Round_Keys[61,0]:=-11348641;
   		Simon_Round_Keys[61,1]:=1941949530;
   		Simon_Round_Keys[62,0]:=1419242898;
   		Simon_Round_Keys[62,1]:=63228607;
   		Simon_Round_Keys[63,0]:=-245036137;
   		Simon_Round_Keys[63,1]:=1400046297;
   		Simon_Round_Keys[64,0]:=-2113955178;
   		Simon_Round_Keys[64,1]:=1642108088;
   		Simon_Round_Keys[65,0]:=1716599554;
   		Simon_Round_Keys[65,1]:=608470937;
   		Simon_Round_Keys[66,0]:=403744995;
   		Simon_Round_Keys[66,1]:=1614638719;
   		Simon_Round_Keys[67,0]:=-585515995;
   		Simon_Round_Keys[67,1]:=-1483187990;
   		Simon_Round_Keys[68,0]:=1561030575;
   		Simon_Round_Keys[68,1]:=1190338945;
   		Simon_Round_Keys[69,0]:=868737890;
   		Simon_Round_Keys[69,1]:=388626190;
   		Simon_Round_Keys[70,0]:=1899935602;
   		Simon_Round_Keys[70,1]:=-2013182834;
   		Simon_Round_Keys[71,0]:=-128145864;
   		Simon_Round_Keys[71,1]:=-999478643;
   End_CASE;
   
END_ROUTINE

ROUTINE SIMON_Rotate_Left1   (* structured text *)
   CASE Simon_Ver Of
   	0:
   		Simon_Rotate_Result[0].[0]:=Simon_tmp2[0].[15];
   		Simon_Rotate_Result[0].[15]:=Simon_tmp2[0].[14];
   		Simon_Rotate_Result[0].[14]:=Simon_tmp2[0].[13];
   		Simon_Rotate_Result[0].[13]:=Simon_tmp2[0].[12];
   		Simon_Rotate_Result[0].[12]:=Simon_tmp2[0].[11];
   		Simon_Rotate_Result[0].[11]:=Simon_tmp2[0].[10];
   		Simon_Rotate_Result[0].[10]:=Simon_tmp2[0].[9];
   		Simon_Rotate_Result[0].[9]:=Simon_tmp2[0].[8];
   		Simon_Rotate_Result[0].[8]:=Simon_tmp2[0].[7];
   		Simon_Rotate_Result[0].[7]:=Simon_tmp2[0].[6];
   		Simon_Rotate_Result[0].[6]:=Simon_tmp2[0].[5];
   		Simon_Rotate_Result[0].[5]:=Simon_tmp2[0].[4];
   		Simon_Rotate_Result[0].[4]:=Simon_tmp2[0].[3];
   		Simon_Rotate_Result[0].[3]:=Simon_tmp2[0].[2];
   		Simon_Rotate_Result[0].[2]:=Simon_tmp2[0].[1];
   		Simon_Rotate_Result[0].[1]:=Simon_tmp2[0].[0];
   	1,2:
   		Simon_Rotate_Result[0].[0]:=Simon_tmp2[0].[31];
   		Simon_Rotate_Result[0].[31]:=Simon_tmp2[0].[30];
   		Simon_Rotate_Result[0].[30]:=Simon_tmp2[0].[29];
   		Simon_Rotate_Result[0].[29]:=Simon_tmp2[0].[28];
   		Simon_Rotate_Result[0].[28]:=Simon_tmp2[0].[27];
   		Simon_Rotate_Result[0].[27]:=Simon_tmp2[0].[26];
   		Simon_Rotate_Result[0].[26]:=Simon_tmp2[0].[25];
   		Simon_Rotate_Result[0].[25]:=Simon_tmp2[0].[24];
   		Simon_Rotate_Result[0].[24]:=Simon_tmp2[0].[23];
   		Simon_Rotate_Result[0].[23]:=Simon_tmp2[0].[22];
   		Simon_Rotate_Result[0].[22]:=Simon_tmp2[0].[21];
   		Simon_Rotate_Result[0].[21]:=Simon_tmp2[0].[20];
   		Simon_Rotate_Result[0].[20]:=Simon_tmp2[0].[19];
   		Simon_Rotate_Result[0].[19]:=Simon_tmp2[0].[18];
   		Simon_Rotate_Result[0].[18]:=Simon_tmp2[0].[17];
   		Simon_Rotate_Result[0].[17]:=Simon_tmp2[0].[16];
   		Simon_Rotate_Result[0].[16]:=Simon_tmp2[0].[15];
   		Simon_Rotate_Result[0].[15]:=Simon_tmp2[0].[14];
   		Simon_Rotate_Result[0].[14]:=Simon_tmp2[0].[13];
   		Simon_Rotate_Result[0].[13]:=Simon_tmp2[0].[12];
   		Simon_Rotate_Result[0].[12]:=Simon_tmp2[0].[11];
   		Simon_Rotate_Result[0].[11]:=Simon_tmp2[0].[10];
   		Simon_Rotate_Result[0].[10]:=Simon_tmp2[0].[9];
   		Simon_Rotate_Result[0].[9]:=Simon_tmp2[0].[8];
   		Simon_Rotate_Result[0].[8]:=Simon_tmp2[0].[7];
   		Simon_Rotate_Result[0].[7]:=Simon_tmp2[0].[6];
   		Simon_Rotate_Result[0].[6]:=Simon_tmp2[0].[5];
   		Simon_Rotate_Result[0].[5]:=Simon_tmp2[0].[4];
   		Simon_Rotate_Result[0].[4]:=Simon_tmp2[0].[3];
   		Simon_Rotate_Result[0].[3]:=Simon_tmp2[0].[2];
   		Simon_Rotate_Result[0].[2]:=Simon_tmp2[0].[1];
   		Simon_Rotate_Result[0].[1]:=Simon_tmp2[0].[0];
   	3,4,5:
   		Simon_Rotate_Result[0].[0]:=Simon_tmp2[1].[31];
   		Simon_Rotate_Result[1].[31]:=Simon_tmp2[1].[30];
   		Simon_Rotate_Result[1].[30]:=Simon_tmp2[1].[29];
   		Simon_Rotate_Result[1].[29]:=Simon_tmp2[1].[28];
   		Simon_Rotate_Result[1].[28]:=Simon_tmp2[1].[27];
   		Simon_Rotate_Result[1].[27]:=Simon_tmp2[1].[26];
   		Simon_Rotate_Result[1].[26]:=Simon_tmp2[1].[25];
   		Simon_Rotate_Result[1].[25]:=Simon_tmp2[1].[24];
   		Simon_Rotate_Result[1].[24]:=Simon_tmp2[1].[23];
   		Simon_Rotate_Result[1].[23]:=Simon_tmp2[1].[22];
   		Simon_Rotate_Result[1].[22]:=Simon_tmp2[1].[21];
   		Simon_Rotate_Result[1].[21]:=Simon_tmp2[1].[20];
   		Simon_Rotate_Result[1].[20]:=Simon_tmp2[1].[19];
   		Simon_Rotate_Result[1].[19]:=Simon_tmp2[1].[18];
   		Simon_Rotate_Result[1].[18]:=Simon_tmp2[1].[17];
   		Simon_Rotate_Result[1].[17]:=Simon_tmp2[1].[16];
   		Simon_Rotate_Result[1].[16]:=Simon_tmp2[1].[15];
   		Simon_Rotate_Result[1].[15]:=Simon_tmp2[1].[14];
   		Simon_Rotate_Result[1].[14]:=Simon_tmp2[1].[13];
   		Simon_Rotate_Result[1].[13]:=Simon_tmp2[1].[12];
   		Simon_Rotate_Result[1].[12]:=Simon_tmp2[1].[11];
   		Simon_Rotate_Result[1].[11]:=Simon_tmp2[1].[10];
   		Simon_Rotate_Result[1].[10]:=Simon_tmp2[1].[9];
   		Simon_Rotate_Result[1].[9]:=Simon_tmp2[1].[8];
   		Simon_Rotate_Result[1].[8]:=Simon_tmp2[1].[7];
   		Simon_Rotate_Result[1].[7]:=Simon_tmp2[1].[6];
   		Simon_Rotate_Result[1].[6]:=Simon_tmp2[1].[5];
   		Simon_Rotate_Result[1].[5]:=Simon_tmp2[1].[4];
   		Simon_Rotate_Result[1].[4]:=Simon_tmp2[1].[3];
   		Simon_Rotate_Result[1].[3]:=Simon_tmp2[1].[2];
   		Simon_Rotate_Result[1].[2]:=Simon_tmp2[1].[1];
   		Simon_Rotate_Result[1].[1]:=Simon_tmp2[1].[0];
   		Simon_Rotate_Result[1].[0]:=Simon_tmp2[0].[31];
   		Simon_Rotate_Result[0].[31]:=Simon_tmp2[0].[30];
   		Simon_Rotate_Result[0].[30]:=Simon_tmp2[0].[29];
   		Simon_Rotate_Result[0].[29]:=Simon_tmp2[0].[28];
   		Simon_Rotate_Result[0].[28]:=Simon_tmp2[0].[27];
   		Simon_Rotate_Result[0].[27]:=Simon_tmp2[0].[26];
   		Simon_Rotate_Result[0].[26]:=Simon_tmp2[0].[25];
   		Simon_Rotate_Result[0].[25]:=Simon_tmp2[0].[24];
   		Simon_Rotate_Result[0].[24]:=Simon_tmp2[0].[23];
   		Simon_Rotate_Result[0].[23]:=Simon_tmp2[0].[22];
   		Simon_Rotate_Result[0].[22]:=Simon_tmp2[0].[21];
   		Simon_Rotate_Result[0].[21]:=Simon_tmp2[0].[20];
   		Simon_Rotate_Result[0].[20]:=Simon_tmp2[0].[19];
   		Simon_Rotate_Result[0].[19]:=Simon_tmp2[0].[18];
   		Simon_Rotate_Result[0].[18]:=Simon_tmp2[0].[17];
   		Simon_Rotate_Result[0].[17]:=Simon_tmp2[0].[16];
   		Simon_Rotate_Result[0].[16]:=Simon_tmp2[0].[15];
   		Simon_Rotate_Result[0].[15]:=Simon_tmp2[0].[14];
   		Simon_Rotate_Result[0].[14]:=Simon_tmp2[0].[13];
   		Simon_Rotate_Result[0].[13]:=Simon_tmp2[0].[12];
   		Simon_Rotate_Result[0].[12]:=Simon_tmp2[0].[11];
   		Simon_Rotate_Result[0].[11]:=Simon_tmp2[0].[10];
   		Simon_Rotate_Result[0].[10]:=Simon_tmp2[0].[9];
   		Simon_Rotate_Result[0].[9]:=Simon_tmp2[0].[8];
   		Simon_Rotate_Result[0].[8]:=Simon_tmp2[0].[7];
   		Simon_Rotate_Result[0].[7]:=Simon_tmp2[0].[6];
   		Simon_Rotate_Result[0].[6]:=Simon_tmp2[0].[5];
   		Simon_Rotate_Result[0].[5]:=Simon_tmp2[0].[4];
   		Simon_Rotate_Result[0].[4]:=Simon_tmp2[0].[3];
   		Simon_Rotate_Result[0].[3]:=Simon_tmp2[0].[2];
   		Simon_Rotate_Result[0].[2]:=Simon_tmp2[0].[1];
   		Simon_Rotate_Result[0].[1]:=Simon_tmp2[0].[0];
   End_CASE;
   
END_ROUTINE

ROUTINE SIMON_Rotate_Left2   (* structured text *)
   CASE Simon_Ver Of
   	0:
   		Simon_Rotate_Result[0].[1]:=Simon_Ciphertext[0,0].[15];
   		Simon_Rotate_Result[0].[0]:=Simon_Ciphertext[0,0].[14];
   		Simon_Rotate_Result[0].[15]:=Simon_Ciphertext[0,0].[13];
   		Simon_Rotate_Result[0].[14]:=Simon_Ciphertext[0,0].[12];
   		Simon_Rotate_Result[0].[13]:=Simon_Ciphertext[0,0].[11];
   		Simon_Rotate_Result[0].[12]:=Simon_Ciphertext[0,0].[10];
   		Simon_Rotate_Result[0].[11]:=Simon_Ciphertext[0,0].[9];
   		Simon_Rotate_Result[0].[10]:=Simon_Ciphertext[0,0].[8];
   		Simon_Rotate_Result[0].[9]:=Simon_Ciphertext[0,0].[7];
   		Simon_Rotate_Result[0].[8]:=Simon_Ciphertext[0,0].[6];
   		Simon_Rotate_Result[0].[7]:=Simon_Ciphertext[0,0].[5];
   		Simon_Rotate_Result[0].[6]:=Simon_Ciphertext[0,0].[4];
   		Simon_Rotate_Result[0].[5]:=Simon_Ciphertext[0,0].[3];
   		Simon_Rotate_Result[0].[4]:=Simon_Ciphertext[0,0].[2];
   		Simon_Rotate_Result[0].[3]:=Simon_Ciphertext[0,0].[1];
   		Simon_Rotate_Result[0].[2]:=Simon_Ciphertext[0,0].[0];
   	1,2:
   		Simon_Rotate_Result[0].[1]:=Simon_tmp2[0].[31];
   		Simon_Rotate_Result[0].[0]:=Simon_tmp2[0].[30];
   		Simon_Rotate_Result[0].[31]:=Simon_tmp2[0].[29];
   		Simon_Rotate_Result[0].[30]:=Simon_tmp2[0].[28];
   		Simon_Rotate_Result[0].[29]:=Simon_tmp2[0].[27];
   		Simon_Rotate_Result[0].[28]:=Simon_tmp2[0].[26];
   		Simon_Rotate_Result[0].[27]:=Simon_tmp2[0].[25];
   		Simon_Rotate_Result[0].[26]:=Simon_tmp2[0].[24];
   		Simon_Rotate_Result[0].[25]:=Simon_tmp2[0].[23];
   		Simon_Rotate_Result[0].[24]:=Simon_tmp2[0].[22];
   		Simon_Rotate_Result[0].[23]:=Simon_tmp2[0].[21];
   		Simon_Rotate_Result[0].[22]:=Simon_tmp2[0].[20];
   		Simon_Rotate_Result[0].[21]:=Simon_tmp2[0].[19];
   		Simon_Rotate_Result[0].[20]:=Simon_tmp2[0].[18];
   		Simon_Rotate_Result[0].[19]:=Simon_tmp2[0].[17];
   		Simon_Rotate_Result[0].[18]:=Simon_tmp2[0].[16];
   		Simon_Rotate_Result[0].[17]:=Simon_tmp2[0].[15];
   		Simon_Rotate_Result[0].[16]:=Simon_tmp2[0].[14];
   		Simon_Rotate_Result[0].[15]:=Simon_tmp2[0].[13];
   		Simon_Rotate_Result[0].[14]:=Simon_tmp2[0].[12];
   		Simon_Rotate_Result[0].[13]:=Simon_tmp2[0].[11];
   		Simon_Rotate_Result[0].[12]:=Simon_tmp2[0].[10];
   		Simon_Rotate_Result[0].[11]:=Simon_tmp2[0].[9];
   		Simon_Rotate_Result[0].[10]:=Simon_tmp2[0].[8];
   		Simon_Rotate_Result[0].[9]:=Simon_tmp2[0].[7];
   		Simon_Rotate_Result[0].[8]:=Simon_tmp2[0].[6];
   		Simon_Rotate_Result[0].[7]:=Simon_tmp2[0].[5];
   		Simon_Rotate_Result[0].[6]:=Simon_tmp2[0].[4];
   		Simon_Rotate_Result[0].[5]:=Simon_tmp2[0].[3];
   		Simon_Rotate_Result[0].[4]:=Simon_tmp2[0].[2];
   		Simon_Rotate_Result[0].[3]:=Simon_tmp2[0].[1];
   		Simon_Rotate_Result[0].[2]:=Simon_tmp2[0].[0];
   	3,4,5:
   		Simon_Rotate_Result[0].[1]:=Simon_tmp2[1].[31];
   		Simon_Rotate_Result[0].[0]:=Simon_tmp2[1].[30];
   		Simon_Rotate_Result[1].[31]:=Simon_tmp2[1].[29];
   		Simon_Rotate_Result[1].[30]:=Simon_tmp2[1].[28];
   		Simon_Rotate_Result[1].[29]:=Simon_tmp2[1].[27];
   		Simon_Rotate_Result[1].[28]:=Simon_tmp2[1].[26];
   		Simon_Rotate_Result[1].[27]:=Simon_tmp2[1].[25];
   		Simon_Rotate_Result[1].[26]:=Simon_tmp2[1].[24];
   		Simon_Rotate_Result[1].[25]:=Simon_tmp2[1].[23];
   		Simon_Rotate_Result[1].[24]:=Simon_tmp2[1].[22];
   		Simon_Rotate_Result[1].[23]:=Simon_tmp2[1].[21];
   		Simon_Rotate_Result[1].[22]:=Simon_tmp2[1].[20];
   		Simon_Rotate_Result[1].[21]:=Simon_tmp2[1].[19];
   		Simon_Rotate_Result[1].[20]:=Simon_tmp2[1].[18];
   		Simon_Rotate_Result[1].[19]:=Simon_tmp2[1].[17];
   		Simon_Rotate_Result[1].[18]:=Simon_tmp2[1].[16];
   		Simon_Rotate_Result[1].[17]:=Simon_tmp2[1].[15];
   		Simon_Rotate_Result[1].[16]:=Simon_tmp2[1].[14];
   		Simon_Rotate_Result[1].[15]:=Simon_tmp2[1].[13];
   		Simon_Rotate_Result[1].[14]:=Simon_tmp2[1].[12];
   		Simon_Rotate_Result[1].[13]:=Simon_tmp2[1].[11];
   		Simon_Rotate_Result[1].[12]:=Simon_tmp2[1].[10];
   		Simon_Rotate_Result[1].[11]:=Simon_tmp2[1].[9];
   		Simon_Rotate_Result[1].[10]:=Simon_tmp2[1].[8];
   		Simon_Rotate_Result[1].[9]:=Simon_tmp2[1].[7];
   		Simon_Rotate_Result[1].[8]:=Simon_tmp2[1].[6];
   		Simon_Rotate_Result[1].[7]:=Simon_tmp2[1].[5];
   		Simon_Rotate_Result[1].[6]:=Simon_tmp2[1].[4];
   		Simon_Rotate_Result[1].[5]:=Simon_tmp2[1].[3];
   		Simon_Rotate_Result[1].[4]:=Simon_tmp2[1].[2];
   		Simon_Rotate_Result[1].[3]:=Simon_tmp2[1].[1];
   		Simon_Rotate_Result[1].[2]:=Simon_tmp2[1].[0];
   		Simon_Rotate_Result[1].[1]:=Simon_tmp2[0].[31];
   		Simon_Rotate_Result[1].[0]:=Simon_tmp2[0].[30];
   		Simon_Rotate_Result[0].[31]:=Simon_tmp2[0].[29];
   		Simon_Rotate_Result[0].[30]:=Simon_tmp2[0].[28];
   		Simon_Rotate_Result[0].[29]:=Simon_tmp2[0].[27];
   		Simon_Rotate_Result[0].[28]:=Simon_tmp2[0].[26];
   		Simon_Rotate_Result[0].[27]:=Simon_tmp2[0].[25];
   		Simon_Rotate_Result[0].[26]:=Simon_tmp2[0].[24];
   		Simon_Rotate_Result[0].[25]:=Simon_tmp2[0].[23];
   		Simon_Rotate_Result[0].[24]:=Simon_tmp2[0].[22];
   		Simon_Rotate_Result[0].[23]:=Simon_tmp2[0].[21];
   		Simon_Rotate_Result[0].[22]:=Simon_tmp2[0].[20];
   		Simon_Rotate_Result[0].[21]:=Simon_tmp2[0].[19];
   		Simon_Rotate_Result[0].[20]:=Simon_tmp2[0].[18];
   		Simon_Rotate_Result[0].[19]:=Simon_tmp2[0].[17];
   		Simon_Rotate_Result[0].[18]:=Simon_tmp2[0].[16];
   		Simon_Rotate_Result[0].[17]:=Simon_tmp2[0].[15];
   		Simon_Rotate_Result[0].[16]:=Simon_tmp2[0].[14];
   		Simon_Rotate_Result[0].[15]:=Simon_tmp2[0].[13];
   		Simon_Rotate_Result[0].[14]:=Simon_tmp2[0].[12];
   		Simon_Rotate_Result[0].[13]:=Simon_tmp2[0].[11];
   		Simon_Rotate_Result[0].[12]:=Simon_tmp2[0].[10];
   		Simon_Rotate_Result[0].[11]:=Simon_tmp2[0].[9];
   		Simon_Rotate_Result[0].[10]:=Simon_tmp2[0].[8];
   		Simon_Rotate_Result[0].[9]:=Simon_tmp2[0].[7];
   		Simon_Rotate_Result[0].[8]:=Simon_tmp2[0].[6];
   		Simon_Rotate_Result[0].[7]:=Simon_tmp2[0].[5];
   		Simon_Rotate_Result[0].[6]:=Simon_tmp2[0].[4];
   		Simon_Rotate_Result[0].[5]:=Simon_tmp2[0].[3];
   		Simon_Rotate_Result[0].[4]:=Simon_tmp2[0].[2];
   		Simon_Rotate_Result[0].[3]:=Simon_tmp2[0].[1];
   		Simon_Rotate_Result[0].[2]:=Simon_tmp2[0].[0];
   End_CASE;
   
END_ROUTINE

ROUTINE SIMON_Rotate_Left8   (* structured text *)
   CASE Simon_Ver Of
   	0:
   		Simon_Rotate_Result[0].[7]:=Simon_Ciphertext[0,0].[15];
   		Simon_Rotate_Result[0].[6]:=Simon_Ciphertext[0,0].[14];
   		Simon_Rotate_Result[0].[5]:=Simon_Ciphertext[0,0].[13];
   		Simon_Rotate_Result[0].[4]:=Simon_Ciphertext[0,0].[12];
   		Simon_Rotate_Result[0].[3]:=Simon_Ciphertext[0,0].[11];
   		Simon_Rotate_Result[0].[2]:=Simon_Ciphertext[0,0].[10];
   		Simon_Rotate_Result[0].[1]:=Simon_Ciphertext[0,0].[9];
   		Simon_Rotate_Result[0].[0]:=Simon_Ciphertext[0,0].[8];
   		Simon_Rotate_Result[0].[15]:=Simon_Ciphertext[0,0].[7];
   		Simon_Rotate_Result[0].[14]:=Simon_Ciphertext[0,0].[6];
   		Simon_Rotate_Result[0].[13]:=Simon_Ciphertext[0,0].[5];
   		Simon_Rotate_Result[0].[12]:=Simon_Ciphertext[0,0].[4];
   		Simon_Rotate_Result[0].[11]:=Simon_Ciphertext[0,0].[3];
   		Simon_Rotate_Result[0].[10]:=Simon_Ciphertext[0,0].[2];
   		Simon_Rotate_Result[0].[9]:=Simon_Ciphertext[0,0].[1];
   		Simon_Rotate_Result[0].[8]:=Simon_Ciphertext[0,0].[0];
   	1,2:
   		Simon_Rotate_Result[0].[7]:=Simon_tmp2[0].[31];
   		Simon_Rotate_Result[0].[6]:=Simon_tmp2[0].[30];
   		Simon_Rotate_Result[0].[5]:=Simon_tmp2[0].[29];
   		Simon_Rotate_Result[0].[4]:=Simon_tmp2[0].[28];
   		Simon_Rotate_Result[0].[3]:=Simon_tmp2[0].[27];
   		Simon_Rotate_Result[0].[2]:=Simon_tmp2[0].[26];
   		Simon_Rotate_Result[0].[1]:=Simon_tmp2[0].[25];
   		Simon_Rotate_Result[0].[0]:=Simon_tmp2[0].[24];
   		Simon_Rotate_Result[0].[31]:=Simon_tmp2[0].[23];
   		Simon_Rotate_Result[0].[30]:=Simon_tmp2[0].[22];
   		Simon_Rotate_Result[0].[29]:=Simon_tmp2[0].[21];
   		Simon_Rotate_Result[0].[28]:=Simon_tmp2[0].[20];
   		Simon_Rotate_Result[0].[27]:=Simon_tmp2[0].[19];
   		Simon_Rotate_Result[0].[26]:=Simon_tmp2[0].[18];
   		Simon_Rotate_Result[0].[25]:=Simon_tmp2[0].[17];
   		Simon_Rotate_Result[0].[24]:=Simon_tmp2[0].[16];
   		Simon_Rotate_Result[0].[23]:=Simon_tmp2[0].[15];
   		Simon_Rotate_Result[0].[22]:=Simon_tmp2[0].[14];
   		Simon_Rotate_Result[0].[21]:=Simon_tmp2[0].[13];
   		Simon_Rotate_Result[0].[20]:=Simon_tmp2[0].[12];
   		Simon_Rotate_Result[0].[19]:=Simon_tmp2[0].[11];
   		Simon_Rotate_Result[0].[18]:=Simon_tmp2[0].[10];
   		Simon_Rotate_Result[0].[17]:=Simon_tmp2[0].[9];
   		Simon_Rotate_Result[0].[16]:=Simon_tmp2[0].[8];
   		Simon_Rotate_Result[0].[15]:=Simon_tmp2[0].[7];
   		Simon_Rotate_Result[0].[14]:=Simon_tmp2[0].[6];
   		Simon_Rotate_Result[0].[13]:=Simon_tmp2[0].[5];
   		Simon_Rotate_Result[0].[12]:=Simon_tmp2[0].[4];
   		Simon_Rotate_Result[0].[11]:=Simon_tmp2[0].[3];
   		Simon_Rotate_Result[0].[10]:=Simon_tmp2[0].[2];
   		Simon_Rotate_Result[0].[9]:=Simon_tmp2[0].[1];
   		Simon_Rotate_Result[0].[8]:=Simon_tmp2[0].[0];
   	3,4,5:
   		Simon_Rotate_Result[0].[7]:=Simon_tmp2[1].[31];
   		Simon_Rotate_Result[0].[6]:=Simon_tmp2[1].[30];
   		Simon_Rotate_Result[0].[5]:=Simon_tmp2[1].[29];
   		Simon_Rotate_Result[0].[4]:=Simon_tmp2[1].[28];
   		Simon_Rotate_Result[0].[3]:=Simon_tmp2[1].[27];
   		Simon_Rotate_Result[0].[2]:=Simon_tmp2[1].[26];
   		Simon_Rotate_Result[0].[1]:=Simon_tmp2[1].[25];
   		Simon_Rotate_Result[0].[0]:=Simon_tmp2[1].[24];
   		Simon_Rotate_Result[1].[31]:=Simon_tmp2[1].[23];
   		Simon_Rotate_Result[1].[30]:=Simon_tmp2[1].[22];
   		Simon_Rotate_Result[1].[29]:=Simon_tmp2[1].[21];
   		Simon_Rotate_Result[1].[28]:=Simon_tmp2[1].[20];
   		Simon_Rotate_Result[1].[27]:=Simon_tmp2[1].[19];
   		Simon_Rotate_Result[1].[26]:=Simon_tmp2[1].[18];
   		Simon_Rotate_Result[1].[25]:=Simon_tmp2[1].[17];
   		Simon_Rotate_Result[1].[24]:=Simon_tmp2[1].[16];
   		Simon_Rotate_Result[1].[23]:=Simon_tmp2[1].[15];
   		Simon_Rotate_Result[1].[22]:=Simon_tmp2[1].[14];
   		Simon_Rotate_Result[1].[21]:=Simon_tmp2[1].[13];
   		Simon_Rotate_Result[1].[20]:=Simon_tmp2[1].[12];
   		Simon_Rotate_Result[1].[19]:=Simon_tmp2[1].[11];
   		Simon_Rotate_Result[1].[18]:=Simon_tmp2[1].[10];
   		Simon_Rotate_Result[1].[17]:=Simon_tmp2[1].[9];
   		Simon_Rotate_Result[1].[16]:=Simon_tmp2[1].[8];
   		Simon_Rotate_Result[1].[15]:=Simon_tmp2[1].[7];
   		Simon_Rotate_Result[1].[14]:=Simon_tmp2[1].[6];
   		Simon_Rotate_Result[1].[13]:=Simon_tmp2[1].[5];
   		Simon_Rotate_Result[1].[12]:=Simon_tmp2[1].[4];
   		Simon_Rotate_Result[1].[11]:=Simon_tmp2[1].[3];
   		Simon_Rotate_Result[1].[10]:=Simon_tmp2[1].[2];
   		Simon_Rotate_Result[1].[9]:=Simon_tmp2[1].[1];
   		Simon_Rotate_Result[1].[8]:=Simon_tmp2[1].[0];
   		Simon_Rotate_Result[1].[7]:=Simon_tmp2[0].[31];
   		Simon_Rotate_Result[1].[6]:=Simon_tmp2[0].[30];
   		Simon_Rotate_Result[1].[5]:=Simon_tmp2[0].[29];
   		Simon_Rotate_Result[1].[4]:=Simon_tmp2[0].[28];
   		Simon_Rotate_Result[1].[3]:=Simon_tmp2[0].[27];
   		Simon_Rotate_Result[1].[2]:=Simon_tmp2[0].[26];
   		Simon_Rotate_Result[1].[1]:=Simon_tmp2[0].[25];
   		Simon_Rotate_Result[1].[0]:=Simon_tmp2[0].[24];
   		Simon_Rotate_Result[0].[31]:=Simon_tmp2[0].[23];
   		Simon_Rotate_Result[0].[30]:=Simon_tmp2[0].[22];
   		Simon_Rotate_Result[0].[29]:=Simon_tmp2[0].[21];
   		Simon_Rotate_Result[0].[28]:=Simon_tmp2[0].[20];
   		Simon_Rotate_Result[0].[27]:=Simon_tmp2[0].[19];
   		Simon_Rotate_Result[0].[26]:=Simon_tmp2[0].[18];
   		Simon_Rotate_Result[0].[25]:=Simon_tmp2[0].[17];
   		Simon_Rotate_Result[0].[24]:=Simon_tmp2[0].[16];
   		Simon_Rotate_Result[0].[23]:=Simon_tmp2[0].[15];
   		Simon_Rotate_Result[0].[22]:=Simon_tmp2[0].[14];
   		Simon_Rotate_Result[0].[21]:=Simon_tmp2[0].[13];
   		Simon_Rotate_Result[0].[20]:=Simon_tmp2[0].[12];
   		Simon_Rotate_Result[0].[19]:=Simon_tmp2[0].[11];
   		Simon_Rotate_Result[0].[18]:=Simon_tmp2[0].[10];
   		Simon_Rotate_Result[0].[17]:=Simon_tmp2[0].[9];
   		Simon_Rotate_Result[0].[16]:=Simon_tmp2[0].[8];
   		Simon_Rotate_Result[0].[15]:=Simon_tmp2[0].[7];
   		Simon_Rotate_Result[0].[14]:=Simon_tmp2[0].[6];
   		Simon_Rotate_Result[0].[13]:=Simon_tmp2[0].[5];
   		Simon_Rotate_Result[0].[12]:=Simon_tmp2[0].[4];
   		Simon_Rotate_Result[0].[11]:=Simon_tmp2[0].[3];
   		Simon_Rotate_Result[0].[10]:=Simon_tmp2[0].[2];
   		Simon_Rotate_Result[0].[9]:=Simon_tmp2[0].[1];
   		Simon_Rotate_Result[0].[8]:=Simon_tmp2[0].[0];
   End_CASE;
   
END_ROUTINE

ROUTINE SIMON_Test   (* structured text *)
   if S:FS then
   	Simon_Ver:=5;     // 0: 32/64, 1: 64: 96, 2: 64:128, 3:128/128, 4:128/192, 5: 128/256
   	//32-64
   	Case Simon_Ver Of
   		0,1,2:
   (*			Simon_Plaintext[0,0]:=26743;  //ver = 0
   			Simon_Plaintext[1,0]:=25957;*)
   
   (*			Simon_Plaintext[0,0]:=1852402787;   //ver = 1
   			Simon_Plaintext[1,0]:=1869750375;*)
   
   			Simon_Plaintext[0,0]:=543452789;    //ver = 2
   			Simon_Plaintext[1,0]:=1701538156;
   
   		3,4,5:
   (*			Simon_Plaintext[0,0]:=1634890784;  //ver = 3
   			Simon_Plaintext[0,1]:=1819043190;
   			Simon_Plaintext[1,0]:=544436837;
   			Simon_Plaintext[1,1]:=1668506980;*)
   
   (*			Simon_Plaintext[0,0]:=1700948338;   //ver = 4
   			Simon_Plaintext[0,1]:=1701345056;
   			Simon_Plaintext[1,0]:=1752440942;
   			Simon_Plaintext[1,1]:=543519333;*)
   
   			Simon_Plaintext[0,0]:=1629516649;
   			Simon_Plaintext[0,1]:=1835627296;   //ver = 5
   			Simon_Plaintext[1,0]:=544042863;
   			Simon_Plaintext[1,1]:=1948282473;
   
   	End_Case;
   	JSR(SIMON_Enc);
   end_if;
   
   
   
   	//JSR(SIMON_Dec);
   
   
END_ROUTINE
END_PROGRAM
